// TIA Portal V20 export
DATA_BLOCK "DB_AxisPosMachinePLC"   // DB103
{ S7_Optimized_Access := 'TRUE' }
// stored: AutoNumber false, MemoryReserve 100
   VAR
      Axis_U1 : Struct
         ExtLoadUnloadAuto : LReal := -3370.0;
         ExtLoadUnloadManu : LReal := -3365.0;
         PartControl : LReal := -3257.0;
         BwLoad : LReal := -1886.83;
         BwUnLoad : LReal := -1962.83;
         BwControl : LReal := -1775.0;
         IntLoadUnload : LReal := -0.2;
         ExtGateExt : LReal := -1164.0;
         IntGateExt : LReal := -857.0;
         ExtGateInt : LReal := -809.0;
         IntGateInt : LReal := -502.0;
         Sas : LReal := -833.0;
         Blowing : LReal := 36.0;
         IntLoadUnloadOP : LReal := 76.0;
      END_STRUCT;
      Axis_U2 : Struct
         ExtLoadUnloadAuto : LReal := -3370.0;
         ExtLoadUnloadManu : LReal := -3365.0;
         PartControl : LReal := -3257.0;
         BwLoad : LReal := -1886.78;
         BwUnLoad : LReal := -1962.78;
         BwControl : LReal := -1775.0;
         IntLoadUnload : LReal := -0.11;
         ExtGateExt : LReal := -1164.0;
         IntGateExt { ExternalAccessible := 'False'; ExternalVisible := 'False'; ExternalWritable := 'False'} : LReal := -857.0;
         ExtGateInt : LReal := -809.0;
         IntGateInt : LReal := -502.0;
         Sas : LReal := -833.0;
         Blowing : LReal := 36.0;
         IntLoadUnloadOP : LReal := 76.0;
      END_STRUCT;
      Axis_V : Struct
         Shuttle_1 : Struct
            LoadUnload : LReal := 17.95;
            Blowing : LReal := 17.95;
         END_STRUCT;
         Shuttle_2 : Struct
            LoadUnload : LReal := -0.48;
            Blowing : LReal := -0.48;
         END_STRUCT;
         Safe : LReal := -0.48;
         Fixture : Struct
            Safe : LReal := 40.0;
            Load : LReal := 192.62;   // 193.52
            Unload : LReal := 192.62;   // 193.52
            Blowing : LReal := 192.62;   // 193.52
         END_STRUCT;
      END_STRUCT;
      Axis_W : Struct
         Shuttle_1 : Struct
            Approach : LReal := -17.61;
            LoadUnload : LReal := -19.61;
            Blowing : LReal := -5.0;
         END_STRUCT;
         Shuttle_2 : Struct
            Approach : LReal := -17.81;
            LoadUnload : LReal := -19.81;
            Blowing : LReal := -5.0;
         END_STRUCT;
         Safe : LReal := 28.5;
         Fixture : Struct
            Safe : LReal := 28.5;
            Load : LReal := -0.8;
            Blowing : LReal := 15.0;
            Unload : LReal := -0.9;
            Approach : LReal := 2.0;
         END_STRUCT;
      END_STRUCT;
   END_VAR
BEGIN
END_DATA_BLOCK
